// TIA Portal project "Pro2" (V16)

(* hardware
DEVICE "S7-1200 station_1"  S7-1200 Station
   slot 0: "Rack_0"  S7-1200 Rack  Rack  V1.0
   slot 1: "PLC_1"  CPU 1214C DC/DC/DC  6ES7 214-1AG40-0XB0  V4.4
   slot 2: "DI 8x24VDC/DQ 8xRelay_1"  SM 1223 DI8/DQ8 x relay  6ES7 223-1PH32-0XB0  V2.0
   slot 3: "AQ 2x14BIT_1"  SM 1232 AQ2  6ES7 232-4HB32-0XB0  V2.1
DEVICE "GSD device_1"  GSD.Device.PN
   slot 0: "机架"  Rack  V1.0
   slot 0: "RobotBasicIO"  BASIC V1.4  888-3  V1.4
      slot 0: "Robot Basic Device"  Robot Basic Device  888-3  V1.4
      slot 1: "PROFINET Interface"  PROFINET Interface
         slot 1: "Network Port"  Network Port
   slot 1: "DI 64 bytes_1"  DI 64 bytes
      slot 0: "DI 64 bytes"  DI 64 bytes
   slot 2: "DO 64 bytes_1"  DO 64 bytes
      slot 0: "DO 64 bytes"  DO 64 bytes
*)

// ===== PLC "PLC_1"  CPU 1214C DC/DC/DC =====
// protected blocks, not shown: "电主轴速度调节", "电主轴速度采集"

VAR_GLOBAL   // PLC tag table "默认变量表"
   "启动按钮" AT %I0.0 : Bool;
   "复位按钮" AT %I0.1 : Bool;
   "换刀信号" AT %I0.2 : Bool;
   "拉刀气压监控" AT %I0.3 : Bool;
   "卸刀气压监控" AT %I0.4 : Bool;
   "拉刀信号反馈" AT %I0.5 : Bool;
   "卸刀信号反馈" AT %I0.6 : Bool;
   "A_7" AT %I0.7 : Bool;
   "U1+" AT %I1.0 : Bool;
   "U1-" AT %I1.1 : Bool;
   "A_10" AT %I1.2 : Bool;
   "A_11" AT %I1.3 : Bool;
   "A_12" AT %I1.4 : Bool;
   "A_13" AT %I1.5 : Bool;
   "变频器停止信号" AT %I2.0 : Bool;
   "变频器启动信号" AT %I2.1 : Bool;
   "A_16" AT %I2.2 : Bool;
   "A_17" AT %I2.3 : Bool;
   "HSC_1_INC" AT %ID1000 : DWord;
   "实时速度输出" AT %QW112 : Int;
   "启动指示灯" AT %Q0.0 : Bool;
   "复位指示灯" AT %Q0.1 : Bool;
   "运行指示灯" AT %Q0.2 : Bool;
   "暂停指示灯" AT %Q0.3 : Bool;
   "故障指示灯" AT %Q0.4 : Bool;
   "拉卸刀电磁阀" AT %Q0.5 : Bool;
   "气源总开关" AT %Q0.6 : Bool;
   "吹尘电磁阀" AT %Q0.7 : Bool;
   "换刀按钮灯" AT %Q1.0 : Bool;
   "B_9" AT %Q1.1 : Bool;
   "System_Byte" AT %MB1 : Byte;
   "FirstScan" AT %M1.0 : Bool;
   "DiagStatusUpdate" AT %M1.1 : Bool;
   "AlwaysTRUE" AT %M1.2 : Bool;
   "AlwaysFALSE" AT %M1.3 : Bool;
   "Clock_Byte" AT %MB0 : Byte;
   "Clock_10Hz" AT %M0.0 : Bool;
   "Clock_5Hz" AT %M0.1 : Bool;
   "Clock_2.5Hz" AT %M0.2 : Bool;
   "Clock_2Hz" AT %M0.3 : Bool;
   "Clock_1.25Hz" AT %M0.4 : Bool;
   "Clock_1Hz" AT %M0.5 : Bool;
   "Clock_0.625Hz" AT %M0.6 : Bool;
   "Clock_0.5Hz" AT %M0.7 : Bool;
   "电主轴启动" AT %M100.0 : Bool;
   "电主轴停止" AT %M100.1 : Bool;
   "电主轴频率递增按钮" AT %M100.2 : Bool;
   "电主轴频率递减按钮" AT %M100.3 : Bool;
   "电主轴运行信号" AT %M100.4 : Bool;
   "电主轴运行指示灯" AT %M100.5 : Bool;
   "HSC_Done" AT %M200.0 : Bool;
   "HSC_Busy" AT %M200.1 : Bool;
   "HSC_Error" AT %M200.2 : Bool;
   "HSC_Status" AT %MW300 : Word;
   "C_4" AT %M200.4 : Bool;
   "C_5" AT %M200.5 : Bool;
   "C_6" AT %M200.6 : Bool;
   "C_7" AT %M200.7 : Bool;
   "GetInteruptData" AT %MD300 : DInt;
   "Frenqucy" AT %MD304 : DInt;
   "Rpm_Second" AT %MD308 : DInt;
   "Rpm_Minute" AT %MD312 : DInt;
   "C_12" AT %MD316 : DInt;
   "C_13" AT %MD320 : DInt;
   "INC_COUNTER" AT %MD1000 : DWord;
   "FromABB" AT %ID100 : DWord;
   "ActualVaule" AT %MD500 : DWord;
   "Tag_1" AT %MW500 : Word;
   "ABB_TO_PLC" AT %I105.0 : Bool;
   "Tag_2" AT %M1100.0 : Bool;
   "换刀" AT %I104.1 : Bool;
   "Tag_3" AT %M1100.1 : Bool;
   "变频器启动" AT %Q10.0 : Bool;
   "变频器停止" AT %Q10.1 : Bool;
   "Tag_4" AT %MD504 : UDInt;
   "R_变频器启动" AT %I104.2 : Bool;
   "R_变频器停止" AT %I104.3 : Bool;
   "R_变频运行" AT %Q2.6 : Bool;
   "Tag_5" AT %M1200.0 : Bool;
   "R_变频停止" AT %Q2.7 : Bool;
END_VAR

TYPE "电机运行及调速控制"
VERSION : 0.1
   STRUCT
      设定运行时间 : Time;
      给定频率 : Real;
   END_STRUCT;
END_TYPE

DATA_BLOCK "Send_HMI_Data"   // DB1
{ S7_Optimized_Access := 'FALSE' }
VERSION : 0.1
   VAR
      Static_1 : Bool;
      Static_2 : Bool;
      电主轴实时转速反馈 : DInt;
      HMI_频率输入 : Real;
      HMI_给定频率 : Real;
   END_VAR
BEGIN
END_DATA_BLOCK

DATA_BLOCK "电主轴运行数据"   // DB2
{ S7_Optimized_Access := 'TRUE' }
VERSION : 0.1
   VAR
      电主轴 : "电机运行及调速控制";
      FromABB : Real;
      FromABBDATA : Array[0..3] of Byte;
      Temp_1 : DWord;
      Temp_2 : DWord;
      Temp_3 : Real;
   END_VAR
BEGIN
END_DATA_BLOCK

DATA_BLOCK "DB_HSC"   // DB3
{ S7_Optimized_Access := 'TRUE' }
VERSION : 0.1
   VAR
      Count : HSC_Count;
   END_VAR
BEGIN
   // Count.CurrentCount : 高速计数器的当前值
   // Count.EnHSC : 启用高速计数器
   // Count.EnSync : 同步输入(I0.7与EnSync同时为1，同步输入才生效)
END_DATA_BLOCK

FUNCTION "气动控制" : Void   // FC1, SCL
{ S7_Optimized_Access := 'TRUE' }
VERSION : 0.1
   VAR_INPUT
      "biTO/TI_Monitor" : Bool;   // 左侧真空压力表
      biCL_Monitor : Bool;   // 右侧压力表
      biTI_SigFeedBack : Bool;   // 拉刀信号反馈
      biTO_SigFeedBack : Bool;   // 卸刀信号反馈
      biExchangeSignal : Bool;   // 换刀信号
      biExchangeSignal_1 : Bool;
   END_VAR
   VAR_OUTPUT
      "boTO/TI" : Bool;   // 拉刀卸刀
      boAirControl : Bool;   // 气源控制
      boCL : Bool;   // 吹尘
      "boTO/TI_Light" : Bool;   // 换刀按钮灯
      boGreenLight : Bool;
      "boRed&buzzer" : Bool;
      boYellowLight : Bool;
   END_VAR
   VAR_TEMP
      T1_OK : Bool;   // 拉刀成功
   END_VAR
BEGIN

   #boAirControl := "AlwaysTRUE";  //开机气源一直为TRUE状态，气封接头一直通气

   //换刀逻辑
   IF #biExchangeSignal OR #biExchangeSignal_1 THEN  //换刀信号为TRUE
       #"boTO/TI" := TRUE;   //换刀电磁阀置1
       #boYellowLight := "Clock_1Hz";
       //#"boRed&buzzer" := "Clock_0.5Hz";
       IF #biTI_SigFeedBack AND NOT #biTO_SigFeedBack THEN//拉刀为TRUE，卸刀为FALSE，换刀成功
           #T1_OK := TRUE; //换刀成功，
       ELSE
           #T1_OK := FALSE;
           #"boRed&buzzer" := "Clock_1Hz";
       END_IF;
   END_IF;


   //中心吹尘
   IF NOT #biTI_SigFeedBack AND #biTO_SigFeedBack THEN
       #boCL := TRUE;
   END_IF;

   IF #biTI_SigFeedBack AND NOT #biTO_SigFeedBack THEN
       #boCL := FALSE;
   END_IF;

   IF NOT #biTI_SigFeedBack AND NOT #biTO_SigFeedBack THEN
       #boYellowLight := "Clock_0.625Hz";
   END_IF;
END_FUNCTION

FUNCTION "报警" : Void   // FC2, SCL
{ S7_Optimized_Access := 'TRUE' }
VERSION : 0.1
   VAR_INPUT
      biTI_Alarm : Bool;
      biTO_Alarm : Bool;
      biReset : Bool;
      biConverter_start : Bool;
   END_VAR
   VAR_OUTPUT
      boRedAlarm : Bool;
   END_VAR
BEGIN
   //压力表报警
   IF #biConverter_start THEN
       IF NOT #biTI_Alarm OR NOT #biTO_Alarm THEN
           #boRedAlarm := TRUE;
       END_IF;
   END_IF;

   IF #biReset THEN
       #boRedAlarm := FALSE;
   END_IF;
END_FUNCTION

ORGANIZATION_BLOCK "Main"   // OB1, LAD, ProgramCycle
TITLE = "Main Program Sweep (Cycle)"
{ S7_Optimized_Access := 'TRUE' }
VERSION : 0.1
   VAR_INPUT
      Initial_Call : Bool;   // Initial call of this OB
      Remanence : Bool;   // =True, if remanent data are available
   END_VAR
BEGIN

REGION Network 1
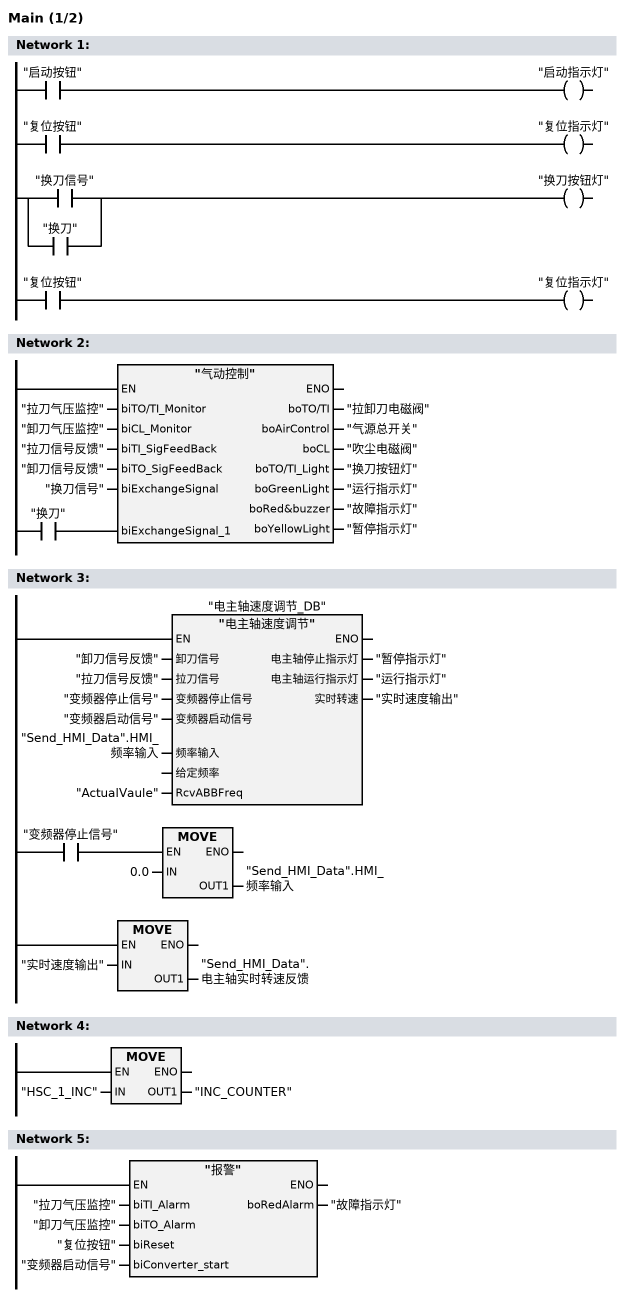
   RUNG wire#powerrail
      Contact( "启动按钮" )
      Coil( "启动指示灯" )
   END_RUNG
   RUNG wire#powerrail
      Contact( "复位按钮" )
      Coil( "复位指示灯" )
   END_RUNG
   RUNG wire#powerrail
      Contact( "换刀信号" )
      wire#w1
      Coil( "换刀按钮灯" )
   END_RUNG
   RUNG wire#powerrail
      Contact( "换刀" )
   END_RUNG wire#w1
   RUNG wire#powerrail
      Contact( "复位按钮" )
      Coil( "复位指示灯" )
   END_RUNG
   // the same network as SCL:
   "启动指示灯" := "启动按钮";
   "复位指示灯" := "复位按钮";
   "换刀按钮灯" := "换刀信号" OR "换刀";
   "复位指示灯" := "复位按钮";
END_REGION

REGION Network 2
   RUNG wire#powerrail
      "气动控制"(biExchangeSignal_1 := wire#w1, "biTO/TI_Monitor" := "拉刀气压监控", biCL_Monitor := "卸刀气压监控", biTI_SigFeedBack := "拉刀信号反馈", biTO_SigFeedBack := "卸刀信号反馈", biExchangeSignal := "换刀信号", "boTO/TI" => "拉卸刀电磁阀", boAirControl => "气源总开关", boCL => "吹尘电磁阀", "boTO/TI_Light" => "换刀按钮灯", boGreenLight => "运行指示灯", "boRed&buzzer" => "故障指示灯", boYellowLight => "暂停指示灯")
   END_RUNG
   RUNG wire#powerrail
      Contact( "换刀" )
   END_RUNG wire#w1
   // the same network as SCL:
   "气动控制"("biTO/TI_Monitor" := "拉刀气压监控",
          biCL_Monitor := "卸刀气压监控",
          biTI_SigFeedBack := "拉刀信号反馈",
          biTO_SigFeedBack := "卸刀信号反馈",
          biExchangeSignal := "换刀信号",
          biExchangeSignal_1 := "换刀",
          "boTO/TI" => "拉卸刀电磁阀",
          boAirControl => "气源总开关",
          boCL => "吹尘电磁阀",
          "boTO/TI_Light" => "换刀按钮灯",
          boGreenLight => "运行指示灯",
          "boRed&buzzer" => "故障指示灯",
          boYellowLight => "暂停指示灯");
END_REGION

REGION Network 3
   RUNG wire#powerrail
      "电主轴速度调节_DB"(卸刀信号 := "卸刀信号反馈", 拉刀信号 := "拉刀信号反馈", 变频器停止信号 := "变频器停止信号", 变频器启动信号 := "变频器启动信号", 频率输入 := "Send_HMI_Data".HMI_频率输入, 给定频率 :=, RcvABBFreq := "ActualVaule", 电主轴停止指示灯 => "暂停指示灯", 电主轴运行指示灯 => "运行指示灯", 实时转速 => "实时速度输出")
   END_RUNG
   RUNG wire#powerrail
      Contact( "变频器停止信号" )
      Move(in := 0.0, out1 => "Send_HMI_Data".HMI_频率输入)
   END_RUNG
   RUNG wire#powerrail
      Move(in := "实时速度输出", out1 => "Send_HMI_Data".电主轴实时转速反馈)
   END_RUNG
   // the same network as SCL:
   "电主轴速度调节_DB"(卸刀信号 := "卸刀信号反馈",   // "电主轴速度调节"
                拉刀信号 := "拉刀信号反馈",
                变频器停止信号 := "变频器停止信号",
                变频器启动信号 := "变频器启动信号",
                频率输入 := "Send_HMI_Data".HMI_频率输入,
                RcvABBFreq := "ActualVaule",
                电主轴停止指示灯 => "暂停指示灯",
                电主轴运行指示灯 => "运行指示灯",
                实时转速 => "实时速度输出");
   IF "变频器停止信号" THEN "Send_HMI_Data".HMI_频率输入 := 0.0; END_IF;
   "Send_HMI_Data".电主轴实时转速反馈 := "实时速度输出";
END_REGION

REGION Network 4
   RUNG wire#powerrail
      Move(in := "HSC_1_INC", out1 => "INC_COUNTER")
   END_RUNG
   // the same network as SCL:
   "INC_COUNTER" := "HSC_1_INC";
END_REGION

REGION Network 5
   RUNG wire#powerrail
      "报警"(biTI_Alarm := "拉刀气压监控", biTO_Alarm := "卸刀气压监控", biReset := "复位按钮", biConverter_start := "变频器启动信号", boRedAlarm => "故障指示灯")
   END_RUNG
   // the same network as SCL:
   "报警"(biTI_Alarm := "拉刀气压监控",
        biTO_Alarm := "卸刀气压监控",
        biReset := "复位按钮",
        biConverter_start := "变频器启动信号",
        boRedAlarm => "故障指示灯");
END_REGION

REGION Network 6
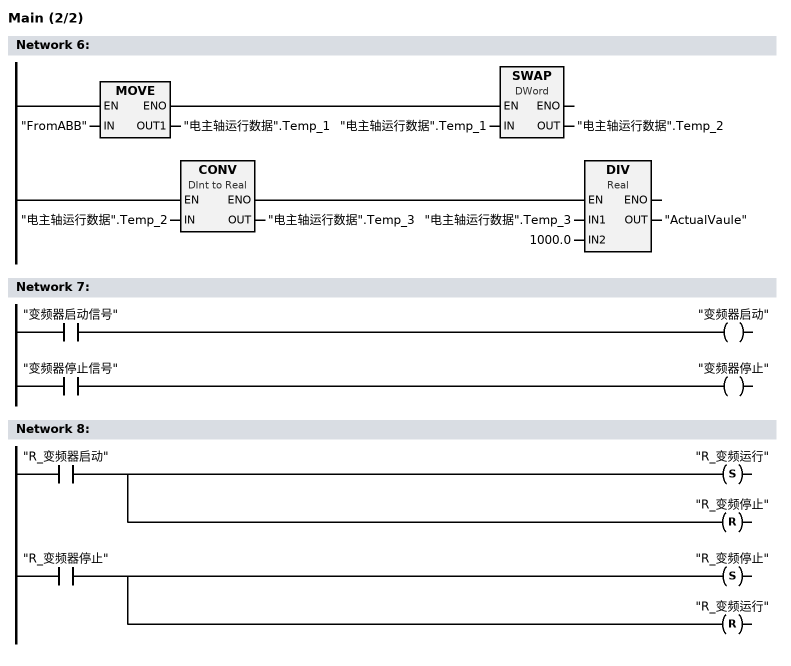
   "电主轴运行数据".Temp_1 := "FromABB";
   "电主轴运行数据".Temp_2 := SWAP("电主轴运行数据".Temp_1);
   "电主轴运行数据".Temp_3 := DINT_TO_REAL("电主轴运行数据".Temp_2);
   "ActualVaule" := "电主轴运行数据".Temp_3 / 1000.0;
END_REGION

REGION Network 7
   RUNG wire#powerrail
      Contact( "变频器启动信号" )
      Coil( "变频器启动" )
   END_RUNG
   RUNG wire#powerrail
      Contact( "变频器停止信号" )
      Coil( "变频器停止" )
   END_RUNG
   // the same network as SCL:
   "变频器启动" := "变频器启动信号";
   "变频器停止" := "变频器停止信号";
END_REGION

REGION Network 8
   RUNG wire#powerrail
      Contact( "R_变频器启动" )
      wire#w1
      S_Coil( "R_变频运行" )
   END_RUNG
   RUNG wire#w1
      R_Coil( "R_变频停止" )
   END_RUNG
   RUNG wire#powerrail
      Contact( "R_变频器停止" )
      wire#w2
      S_Coil( "R_变频停止" )
   END_RUNG
   RUNG wire#w2
      R_Coil( "R_变频运行" )
   END_RUNG
   // the same network as SCL:
   IF "R_变频器启动" THEN
       "R_变频运行" := TRUE;
       "R_变频停止" := FALSE;
   END_IF;
   IF "R_变频器停止" THEN
       "R_变频停止" := TRUE;
       "R_变频运行" := FALSE;
   END_IF;
END_REGION
END_ORGANIZATION_BLOCK

ORGANIZATION_BLOCK "Cyclic interrupt"   // OB30, LAD, CyclicInterrupt
{ S7_Optimized_Access := 'TRUE' }
VERSION : 0.1
   VAR_INPUT
      Initial_Call : Bool;   // Initial call of this OB
      Event_Count : Int;   // Events discarded
   END_VAR
BEGIN

REGION Network 1
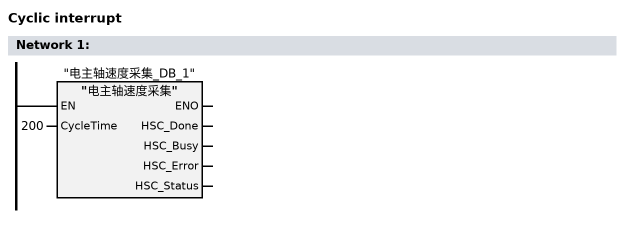
   RUNG wire#powerrail
      "电主轴速度采集_DB_1"(CycleTime := 200, HSC_Done =>, HSC_Busy =>, HSC_Error =>, HSC_Status =>)
   END_RUNG
   // the same network as SCL:
   "电主轴速度采集_DB_1"(CycleTime := 200);   // "电主轴速度采集"
END_REGION
END_ORGANIZATION_BLOCK

ORGANIZATION_BLOCK "Hardware interrupt"   // OB40, LAD, HWProcessInterrupt
{ S7_Optimized_Access := 'TRUE' }
VERSION : 0.1
   VAR_INPUT
      LADDR : Hw_Io;   // Hardware identifier
      USI : Word;   // User structure identifier
      IChannel : USInt;   // Interrupt channel number
      EventType : Byte;   // EventType
   END_VAR
BEGIN
END_ORGANIZATION_BLOCK